{attribute 'enable_dynamic_creation'}
FUNCTION_BLOCK FutureMCHalt EXTENDS FB_AbstructFuture
VAR_INPUT
END_VAR
VAR_OUTPUT
END_VAR
VAR
	_axis: REFERENCE TO AXIS_REF;
	_fb_halt	: MC_Halt;
	_mc_reset	: MC_Reset;
	_deceleration: MC_LREAL;
	_jerk		: MC_LREAL;
	_option : ST_MoveOptions;
	_buffer_mode : MC_BufferMode;
	_error_id :HRESULT;
	_exec_state : UDINT;
END_VAR

METHOD error_reset : BOOL // Must be overrided if future has any errors.
IF _error_id <> 0 THEN
	CASE _exec_state OF
		0:
			_mc_reset(Axis := _axis, Execute := FALSE);
			_mc_reset(Axis:= _axis, Execute := TRUE );
			_exec_state := 1;
		1:
			IF _mc_reset.Busy THEN
				_mc_reset(Axis:= _axis,Execute := FALSE);
			END_IF
	END_CASE
	
	_error_id := _mc_reset.ErrorID;
	error_reset := _mc_reset.Done;
ELSE
	error_reset := TRUE;
END_IF
END_METHOD

METHOD execute : BOOL // Return TRUE if finish.

CASE _exec_state OF
	0:
		_fb_halt(axis := _axis, Execute := FALSE);
		_fb_halt(
			Axis:= _axis,
			Execute := TRUE,
			Jerk := _jerk,
			BufferMode := _buffer_mode,
			Options := _option
		);
		_exec_state := 1;
	1:
		IF _fb_halt.Busy THEN
			_fb_halt(Axis:= _axis,Execute := FALSE);
		END_IF
END_CASE

_error_id := _fb_halt.ErrorID;
execute := _fb_halt.Done OR _fb_halt.Error;
END_METHOD

METHOD init : BOOL // Return TRUE if finish.
_exec_state := 0;
init := TRUE;
END_METHOD

PROPERTY nErrorID : HRESULT
GET
nErrorID := _error_id;
END_GET
SET
END_SET
END_PROPERTY

METHOD set_options : BOOL
VAR_INPUT
	buffer_mode : MC_BufferMode;
	option : ST_MoveOptions;
END_VAR
_buffer_mode := buffer_mode;
_option := option;
END_METHOD

METHOD set_parameters : BOOL
VAR_INPUT
	axis : REFERENCE TO AXIS_REF;
	deceleration	: MC_LREAL;		// Set deceleration in case let moving axis halt.
	jerk			: MC_LREAL;		// Set jerk in case let moving axis halt.
END_VAR
_axis REF= axis;
_deceleration := deceleration;
_jerk := jerk;
END_METHOD

END_FUNCTION_BLOCK

(* stored: Version 1.1.0.1, ProductVersion 3.1.4026.13
   POU FutureMCHalt: Id {2dc714ff-adc1-44ab-b7e0-76a95eea807d}, SpecialFunc None
   Method error_reset: Id {207df50c-02d9-4f34-a222-e45f864c0020}
   Method execute: Id {fb168655-c2e0-4f32-bbeb-489e0cb4dd0f}
   Method init: Id {ffd4fbac-b56b-4623-94bb-267c8989ec1e}
   Property nErrorID: Id {f26f4ea7-8ce7-49fa-9833-3e578be10865}
   Get Get: Id {4fb1eb75-3038-4c58-a8ee-43f876083f46}
   Set Set: Id {6d9612dd-335e-4051-9373-3a34dde3e997}
   Method set_options: Id {4a63d360-82fa-4437-aeca-057b879f625c}
   Method set_parameters: Id {8b458c83-829b-4614-8ee0-e4ba57723626} *)
